FUNCTION_BLOCK FB_ReferenceManager
VAR_OUTPUT
	Error : BOOL;
	ErrorMessage : STRING(255);
END_VAR
VAR
	_Names : ARRAY[1..Param_Config.MaxConfigReferenceNodes] OF STRING(255);
	_BaseUnits : ARRAY[1..Param_Config.MaxConfigReferenceNodes] OF I_BaseUnit;
	_Count : UINT;
END_VAR

METHOD PUBLIC M_RegisterReference : BOOL
VAR_INPUT
	Name : STRING(255);
	BaseUnit : I_BaseUnit;
END_VAR
VAR
	nIndex : UINT;
END_VAR
M_RegisterReference := FALSE;
Error := FALSE;
ErrorMessage := '';
IF BaseUnit = 0 THEN
	Error := TRUE;
	ErrorMessage := 'Cannot register an unbound BaseUnit interface.';
	RETURN;
END_IF

FOR nIndex := 1 TO _Count DO
	IF _Names[nIndex] = Name THEN
		_BaseUnits[nIndex] := BaseUnit;
		M_RegisterReference := TRUE;
		RETURN;
	END_IF
END_FOR

nIndex := _Count + 1;
IF nIndex > Param_Config.MaxConfigReferenceNodes THEN
	Error := TRUE;
	ErrorMessage := 'Reference registry is full.';
	RETURN;
END_IF

_Names[nIndex] := Name;
_BaseUnits[nIndex] := BaseUnit;
_Count := nIndex;
M_RegisterReference := TRUE;
END_METHOD

METHOD PUBLIC M_Resolve : I_BaseUnit
VAR_INPUT
	Name : STRING(255);
END_VAR
VAR
	nIndex : UINT;
END_VAR
M_Resolve := 0;
Error := FALSE;
ErrorMessage := '';
FOR nIndex := 1 TO _Count DO
	IF _Names[nIndex] = Name THEN
		M_Resolve := _BaseUnits[nIndex];
		RETURN;
	END_IF
END_FOR
Error := TRUE;
ErrorMessage := 'Reference source was not registered.';
END_METHOD

END_FUNCTION_BLOCK

(* stored: Version 1.1.0.1, ProductVersion 3.1.4026.18
   POU FB_ReferenceManager: Id {9876fc16-fe16-4cc5-b330-d893d8344748}, SpecialFunc None
   Method M_RegisterReference: Id {30f6847e-f317-4205-a8d3-568bd3a0a3e6}
   Method M_Resolve: Id {846010cd-2d2e-466c-a333-6b11259411bc} *)
